{attribute addProperty BoxType "EL1252-0000-0017"}
{attribute addProperty Id "Status0AT %I*USINT81174Status1AT %I*USINT81175LatchPos0AT %I*ULINT648176LatchNeg0AT %I*ULINT648184LatchPos1AT %I*ULINT648192LatchNeg1AT %I*ULINT648200"}
{attribute addProperty CRC "1423568066"}
{attribute addProperty SizeInBites "272"}
{attribute addProperty SizeInBytes "34"}
TYPE Latch_54D9ECC2 :
STRUCT
	{attribute addProperty Name "Status0"}
	Status0 AT %I* : USINT;
	{attribute addProperty Name "Status1"}
	Status1 AT %I* : USINT;
	{attribute addProperty Name "LatchPos0"}
	LatchPos0 AT %I* : ULINT;
	{attribute addProperty Name "LatchNeg0"}
	LatchNeg0 AT %I* : ULINT;
	{attribute addProperty Name "LatchPos1"}
	LatchPos1 AT %I* : ULINT;
	{attribute addProperty Name "LatchNeg1"}
	LatchNeg1 AT %I* : ULINT;
END_STRUCT
END_TYPE

(* stored: Version 1.2.0.0, ProductVersion 3.1.4024.9
   DUT Latch_54D9ECC2: Id {4ac8084c-4ebd-4fc1-83ee-e70efd6ffa57} *)
